INTERFACE I_Mc3Axis EXTENDS I_Component, I_AxisEnable, I_Mc3AxisRef, I_Resettable, I_Stoppable, I_AxisDynamics, I_AxisStatus, I_AxisJog, I_AxisHome, I_Mc3Settings, I_Override

{attribute 'monitoring' := 'call'}
PROPERTY ErrorId : UDINT
GET
END_GET
END_PROPERTY

PROPERTY MotionTasks : I_Mc3MotionTaskCollection
GET
END_GET
END_PROPERTY

END_INTERFACE

(* stored: Version 1.1.0.1, ProductVersion 3.1.4026.20
   Itf I_Mc3Axis: Id {fb36648c-4ae2-4934-a09b-d28e9229474b}
   Property ErrorId: Id {a0d3ec5b-eae4-4799-ae19-283af281757b}
   Get Get: Id {876ae65a-9ba8-42b8-9eed-5be72f5fa06e}
   Property MotionTasks: Id {d7b355c1-3564-4cfa-9ece-89a01977069e}
   Get Get: Id {09373c36-c698-4846-ad60-f1e55ef265b4} *)
